FUNCTION_BLOCK FB_BA_Umschaltung_FUP
VAR_INPUT
END_VAR
VAR_OUTPUT
END_VAR
VAR
	FB_BA_Hand : FB_Betriebsarten;
	FB_BA_Auto : FB_Betriebsarten;
END_VAR

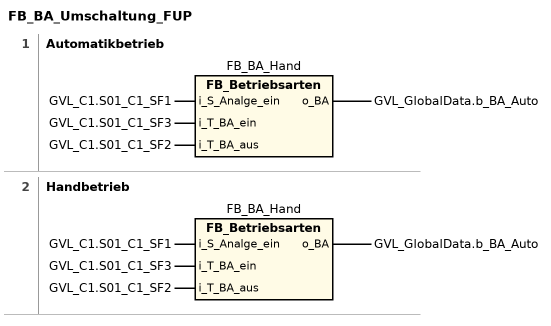
// NETWORK 1: Automatikbetrieb
FB_BA_Hand(
    i_S_Analge_ein := GVL_C1.S01_C1_SF1,
    i_T_BA_ein := GVL_C1.S01_C1_SF3,
    i_T_BA_aus := GVL_C1.S01_C1_SF2); // FB_Betriebsarten
GVL_GlobalData.b_BA_Auto := FB_BA_Hand.o_BA;

// NETWORK 2: Handbetrieb
FB_BA_Hand(
    i_S_Analge_ein := GVL_C1.S01_C1_SF1,
    i_T_BA_ein := GVL_C1.S01_C1_SF3,
    i_T_BA_aus := GVL_C1.S01_C1_SF2); // FB_Betriebsarten
GVL_GlobalData.b_BA_Auto := FB_BA_Hand.o_BA;

END_FUNCTION_BLOCK

(* stored: Version 1.1.0.1, ProductVersion 3.1.4024.12
   POU FB_BA_Umschaltung_FUP: Id {c39b4d99-11ad-4205-97de-ef62c6bda110}, SpecialFunc None *)
